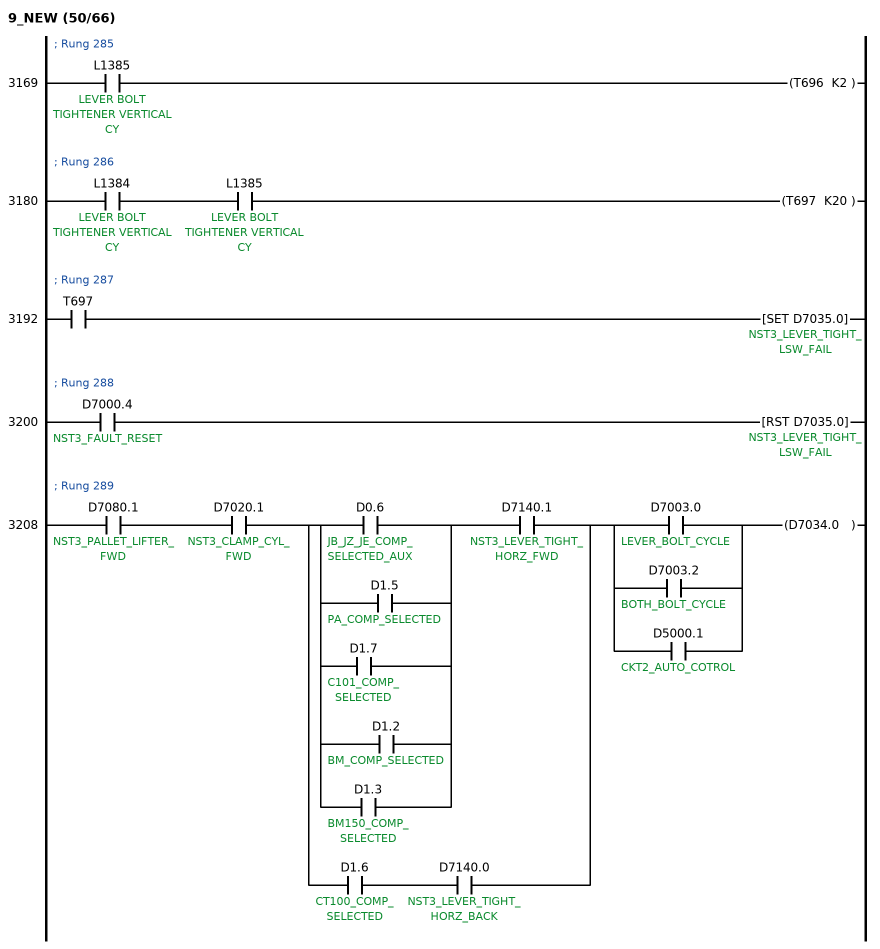
[picture p168: ladder of 9_NEW, rungs at steps 3169 to 3208]
; Rung 285
3169  LD      L1385  ; LEVER BOLT TIGHTENER VERTICAL CY
      OUT     T696 K2
; Rung 286
3180  LD      L1384  ; LEVER BOLT TIGHTENER VERTICAL CY
      AND     L1385  ; LEVER BOLT TIGHTENER VERTICAL CY
      OUT     T697 K20
; Rung 287
3192  LD      T697
      SET     D7035.0  ; NST3_LEVER_TIGHT_LSW_FAIL
; Rung 288
3200  LD      D7000.4  ; NST3_FAULT_RESET
      RST     D7035.0  ; NST3_LEVER_TIGHT_LSW_FAIL
; Rung 289
3208  LD      D7080.1  ; NST3_PALLET_LIFTER_FWD
      AND     D7020.1  ; NST3_CLAMP_CYL_FWD
      LD      D0.6  ; JB_JZ_JE_COMP_SELECTED_AUX
      OR      D1.5  ; PA_COMP_SELECTED
      OR      D1.7  ; C101_COMP_SELECTED
      OR      D1.2  ; BM_COMP_SELECTED
      OR      D1.3  ; BM150_COMP_SELECTED
      AND     D7140.1  ; NST3_LEVER_TIGHT_HORZ_FWD
      LD      D1.6  ; CT100_COMP_SELECTED
      AND     D7140.0  ; NST3_LEVER_TIGHT_HORZ_BACK
      ORB
      ANB
      LD      D7003.0  ; LEVER_BOLT_CYCLE
      OR      D7003.2  ; BOTH_BOLT_CYCLE
      OR      D5000.1  ; CKT2_AUTO_COTROL
      ANB
      OUT     D7034.0
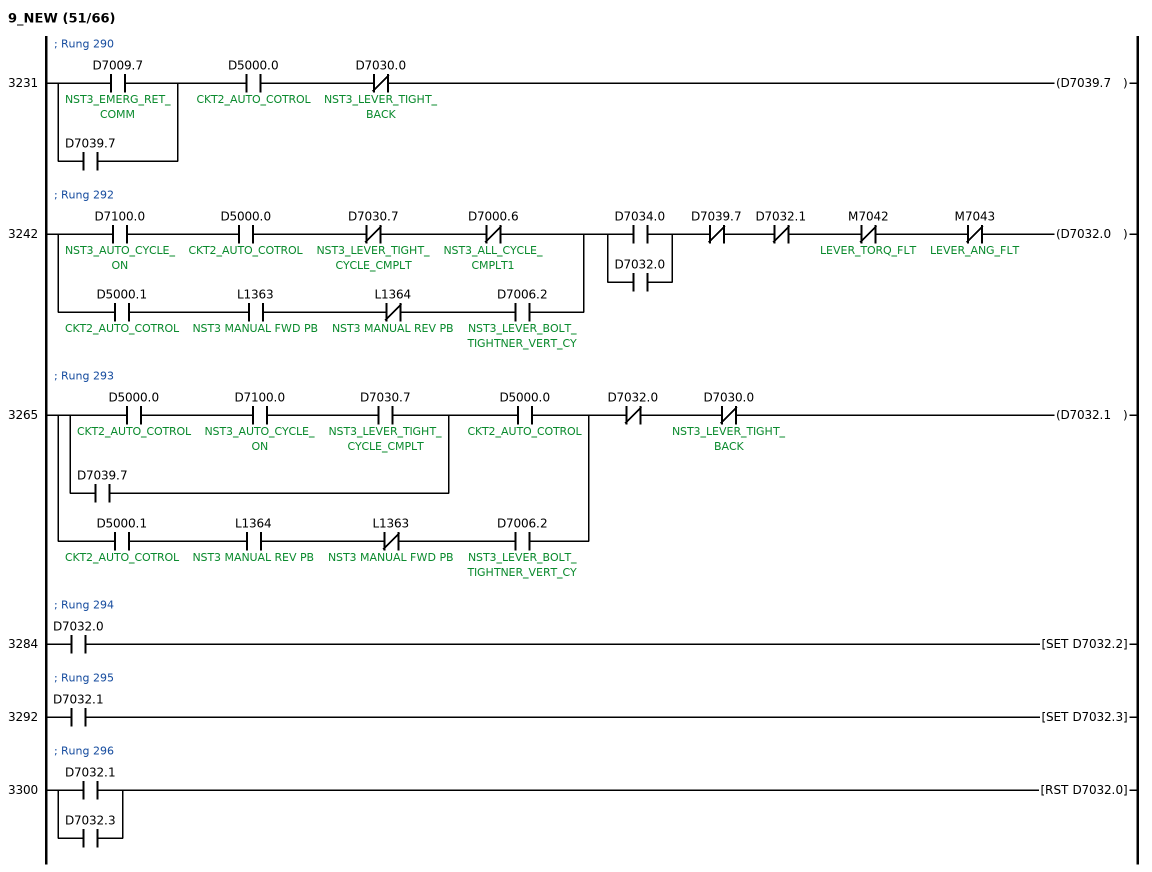
; Rung 290
3231  LD      D7009.7  ; NST3_EMERG_RET_COMM
      OR      D7039.7
      AND     D5000.0  ; CKT2_AUTO_COTROL
      ANI     D7030.0  ; NST3_LEVER_TIGHT_BACK
      OUT     D7039.7
; Rung 292
3242  LD      D7100.0  ; NST3_AUTO_CYCLE_ON
      AND     D5000.0  ; CKT2_AUTO_COTROL
      ANI     D7030.7  ; NST3_LEVER_TIGHT_CYCLE_CMPLT
      ANI     D7000.6  ; NST3_ALL_CYCLE_CMPLT1
      LD      D5000.1  ; CKT2_AUTO_COTROL
      AND     L1363  ; NST3 MANUAL FWD PB
      ANI     L1364  ; NST3 MANUAL REV PB
      AND     D7006.2  ; NST3_LEVER_BOLT_TIGHTNER_VERT_CY
      ORB
      LD      D7034.0
      OR      D7032.0
      ANB
      ANI     D7039.7
      ANI     D7032.1
      ANI     M7042  ; LEVER_TORQ_FLT
      ANI     M7043  ; LEVER_ANG_FLT
      OUT     D7032.0
; Rung 293
3265  LD      D5000.0  ; CKT2_AUTO_COTROL
      AND     D7100.0  ; NST3_AUTO_CYCLE_ON
      AND     D7030.7  ; NST3_LEVER_TIGHT_CYCLE_CMPLT
      OR      D7039.7
      AND     D5000.0  ; CKT2_AUTO_COTROL
      LD      D5000.1  ; CKT2_AUTO_COTROL
      AND     L1364  ; NST3 MANUAL REV PB
      ANI     L1363  ; NST3 MANUAL FWD PB
      AND     D7006.2  ; NST3_LEVER_BOLT_TIGHTNER_VERT_CY
      ORB
      ANI     D7032.0
      ANI     D7030.0  ; NST3_LEVER_TIGHT_BACK
      OUT     D7032.1
; Rung 294
3284  LD      D7032.0
      SET     D7032.2
; Rung 295
3292  LD      D7032.1
      SET     D7032.3
; Rung 296
3300  LD      D7032.1
      OR      D7032.3
      RST     D7032.0
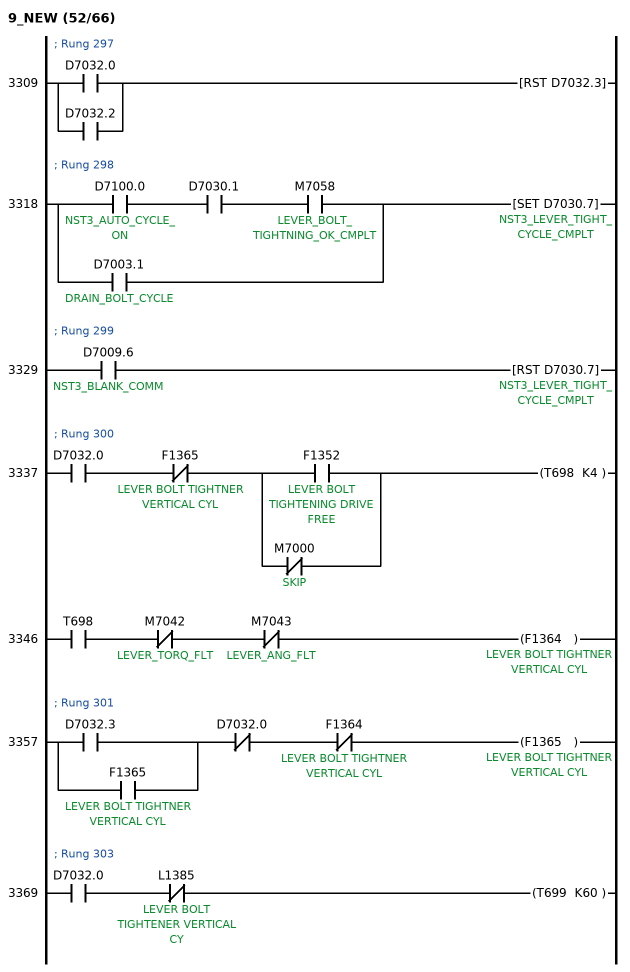
; Rung 297
3309  LD      D7032.0
      OR      D7032.2
      RST     D7032.3
; Rung 298
3318  LD      D7100.0  ; NST3_AUTO_CYCLE_ON
      AND     D7030.1
      AND     M7058  ; LEVER_BOLT_TIGHTNING_OK_CMPLT
      OR      D7003.1  ; DRAIN_BOLT_CYCLE
      SET     D7030.7  ; NST3_LEVER_TIGHT_CYCLE_CMPLT
; Rung 299
3329  LD      D7009.6  ; NST3_BLANK_COMM
      RST     D7030.7  ; NST3_LEVER_TIGHT_CYCLE_CMPLT
; Rung 300
3337  LD      D7032.0
      ANI     F1365  ; LEVER BOLT TIGHTNER VERTICAL CYL
      LD      F1352  ; LEVER BOLT TIGHTENING DRIVE FREE
      ORI     M7000  ; SKIP
      ANB
      OUT     T698 K4
3346  LD      T698
      ANI     M7042  ; LEVER_TORQ_FLT
      ANI     M7043  ; LEVER_ANG_FLT
      OUT     F1364  ; LEVER BOLT TIGHTNER VERTICAL CYL
; Rung 301
3357  LD      D7032.3
      OR      F1365  ; LEVER BOLT TIGHTNER VERTICAL CYL
      ANI     D7032.0
      ANI     F1364  ; LEVER BOLT TIGHTNER VERTICAL CYL
      OUT     F1365  ; LEVER BOLT TIGHTNER VERTICAL CYL
; Rung 303
3369  LD      D7032.0
      ANI     L1385  ; LEVER BOLT TIGHTENER VERTICAL CY
      OUT     T699 K60
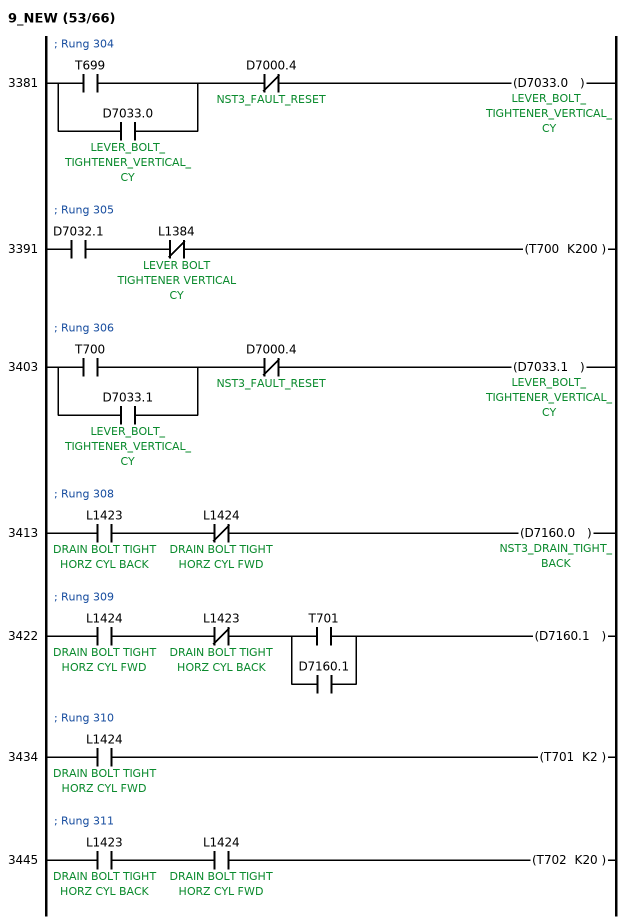
; Rung 304
3381  LD      T699
      OR      D7033.0  ; LEVER_BOLT_TIGHTENER_VERTICAL_CY
      ANI     D7000.4  ; NST3_FAULT_RESET
      OUT     D7033.0  ; LEVER_BOLT_TIGHTENER_VERTICAL_CY
; Rung 305
3391  LD      D7032.1
      ANI     L1384  ; LEVER BOLT TIGHTENER VERTICAL CY
      OUT     T700 K200
; Rung 306
3403  LD      T700
      OR      D7033.1  ; LEVER_BOLT_TIGHTENER_VERTICAL_CY
      ANI     D7000.4  ; NST3_FAULT_RESET
      OUT     D7033.1  ; LEVER_BOLT_TIGHTENER_VERTICAL_CY
; Rung 308
3413  LD      L1423  ; DRAIN BOLT TIGHT HORZ CYL BACK
      ANI     L1424  ; DRAIN BOLT TIGHT HORZ CYL FWD
      OUT     D7160.0  ; NST3_DRAIN_TIGHT_BACK
; Rung 309
3422  LD      L1424  ; DRAIN BOLT TIGHT HORZ CYL FWD
      ANI     L1423  ; DRAIN BOLT TIGHT HORZ CYL BACK
      LD      T701
      OR      D7160.1
      ANB
      OUT     D7160.1
; Rung 310
3434  LD      L1424  ; DRAIN BOLT TIGHT HORZ CYL FWD
      OUT     T701 K2
; Rung 311
3445  LD      L1423  ; DRAIN BOLT TIGHT HORZ CYL BACK
      AND     L1424  ; DRAIN BOLT TIGHT HORZ CYL FWD
      OUT     T702 K20
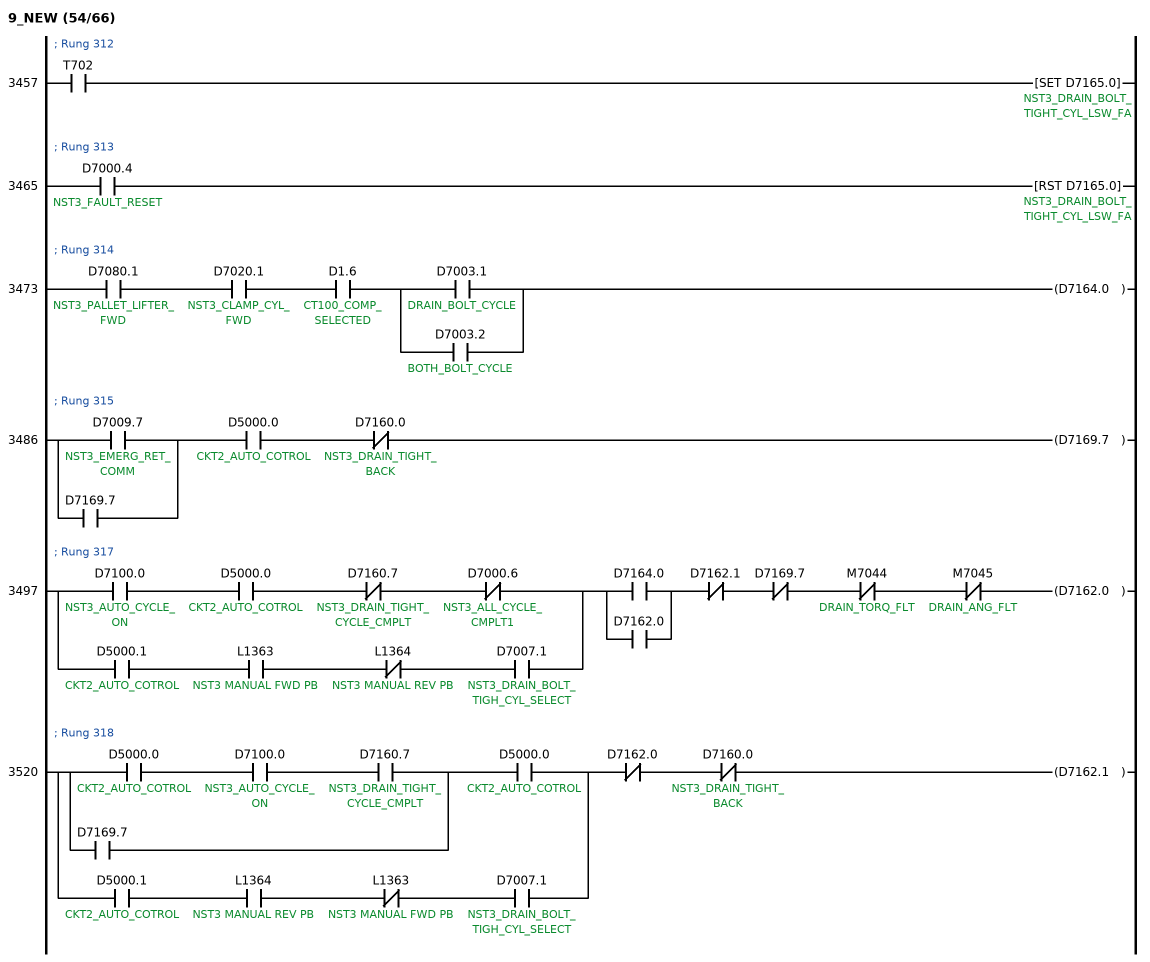
; Rung 312
3457  LD      T702
      SET     D7165.0  ; NST3_DRAIN_BOLT_TIGHT_CYL_LSW_FA
; Rung 313
3465  LD      D7000.4  ; NST3_FAULT_RESET
      RST     D7165.0  ; NST3_DRAIN_BOLT_TIGHT_CYL_LSW_FA
; Rung 314
3473  LD      D7080.1  ; NST3_PALLET_LIFTER_FWD
      AND     D7020.1  ; NST3_CLAMP_CYL_FWD
      AND     D1.6  ; CT100_COMP_SELECTED
      LD      D7003.1  ; DRAIN_BOLT_CYCLE
      OR      D7003.2  ; BOTH_BOLT_CYCLE
      ANB
      OUT     D7164.0
; Rung 315
3486  LD      D7009.7  ; NST3_EMERG_RET_COMM
      OR      D7169.7
      AND     D5000.0  ; CKT2_AUTO_COTROL
      ANI     D7160.0  ; NST3_DRAIN_TIGHT_BACK
      OUT     D7169.7
; Rung 317
3497  LD      D7100.0  ; NST3_AUTO_CYCLE_ON
      AND     D5000.0  ; CKT2_AUTO_COTROL
      ANI     D7160.7  ; NST3_DRAIN_TIGHT_CYCLE_CMPLT
      ANI     D7000.6  ; NST3_ALL_CYCLE_CMPLT1
      LD      D5000.1  ; CKT2_AUTO_COTROL
      AND     L1363  ; NST3 MANUAL FWD PB
      ANI     L1364  ; NST3 MANUAL REV PB
      AND     D7007.1  ; NST3_DRAIN_BOLT_TIGH_CYL_SELECT
      ORB
      LD      D7164.0
      OR      D7162.0
      ANB
      ANI     D7162.1
      ANI     D7169.7
      ANI     M7044  ; DRAIN_TORQ_FLT
      ANI     M7045  ; DRAIN_ANG_FLT
      OUT     D7162.0
; Rung 318
3520  LD      D5000.0  ; CKT2_AUTO_COTROL
      AND     D7100.0  ; NST3_AUTO_CYCLE_ON
      AND     D7160.7  ; NST3_DRAIN_TIGHT_CYCLE_CMPLT
      OR      D7169.7
      AND     D5000.0  ; CKT2_AUTO_COTROL
      LD      D5000.1  ; CKT2_AUTO_COTROL
      AND     L1364  ; NST3 MANUAL REV PB
      ANI     L1363  ; NST3 MANUAL FWD PB
      AND     D7007.1  ; NST3_DRAIN_BOLT_TIGH_CYL_SELECT
      ORB
      ANI     D7162.0
      ANI     D7160.0  ; NST3_DRAIN_TIGHT_BACK
      OUT     D7162.1
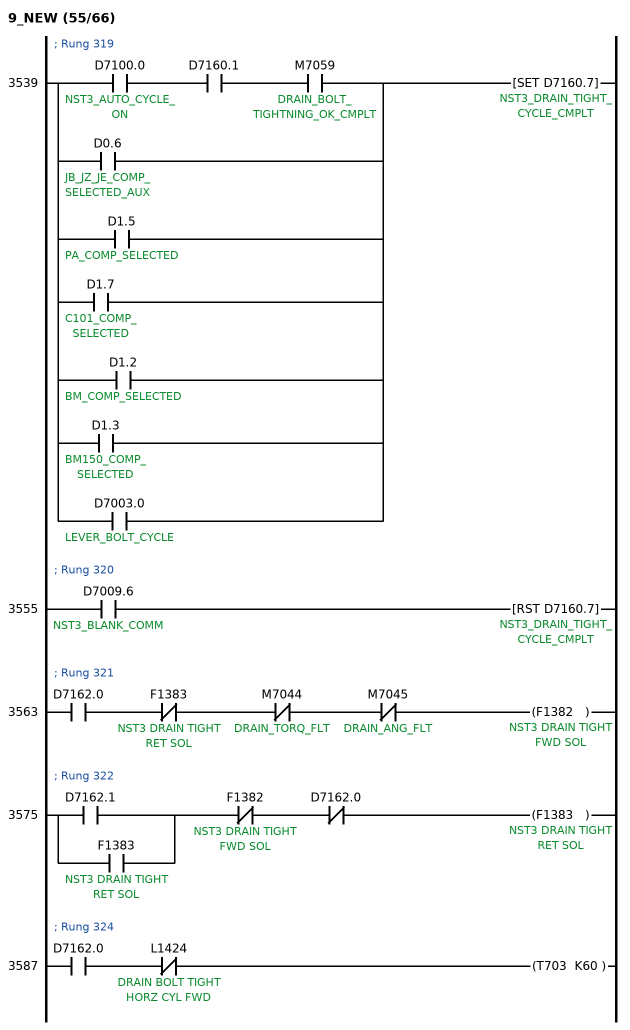
; Rung 319
3539  LD      D7100.0  ; NST3_AUTO_CYCLE_ON
      AND     D7160.1
      AND     M7059  ; DRAIN_BOLT_TIGHTNING_OK_CMPLT
      OR      D0.6  ; JB_JZ_JE_COMP_SELECTED_AUX
      OR      D1.5  ; PA_COMP_SELECTED
      OR      D1.7  ; C101_COMP_SELECTED
      OR      D1.2  ; BM_COMP_SELECTED
      OR      D1.3  ; BM150_COMP_SELECTED
      OR      D7003.0  ; LEVER_BOLT_CYCLE
      SET     D7160.7  ; NST3_DRAIN_TIGHT_CYCLE_CMPLT
; Rung 320
3555  LD      D7009.6  ; NST3_BLANK_COMM
      RST     D7160.7  ; NST3_DRAIN_TIGHT_CYCLE_CMPLT
; Rung 321
3563  LD      D7162.0
      ANI     F1383  ; NST3 DRAIN TIGHT RET SOL
      ANI     M7044  ; DRAIN_TORQ_FLT
      ANI     M7045  ; DRAIN_ANG_FLT
      OUT     F1382  ; NST3 DRAIN TIGHT FWD SOL
; Rung 322
3575  LD      D7162.1
      OR      F1383  ; NST3 DRAIN TIGHT RET SOL
      ANI     F1382  ; NST3 DRAIN TIGHT FWD SOL
      ANI     D7162.0
      OUT     F1383  ; NST3 DRAIN TIGHT RET SOL
; Rung 324
3587  LD      D7162.0
      ANI     L1424  ; DRAIN BOLT TIGHT HORZ CYL FWD
      OUT     T703 K60
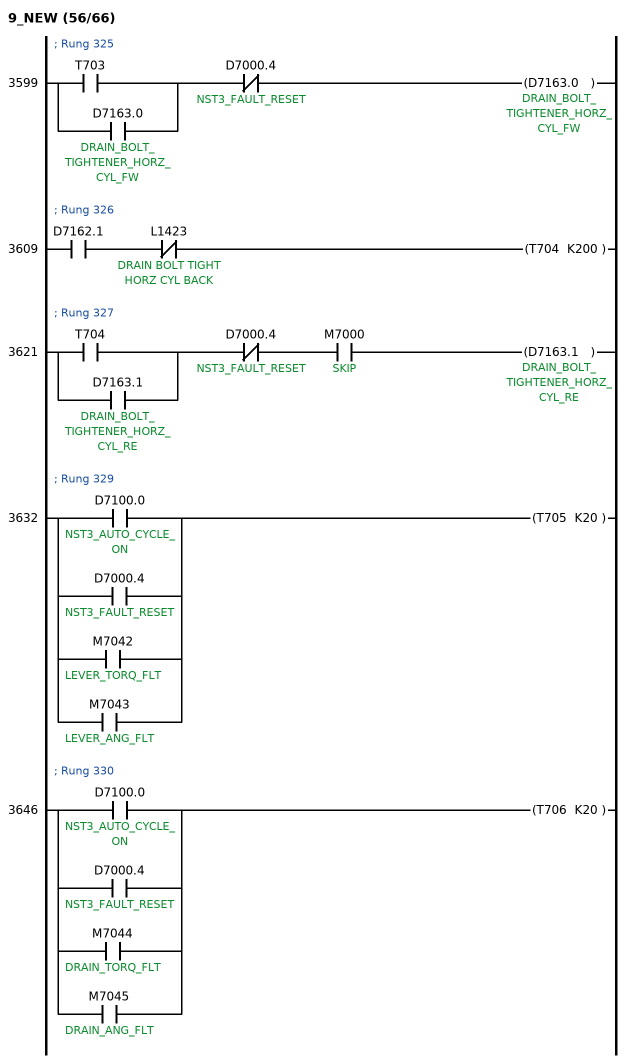
; Rung 325
3599  LD      T703
      OR      D7163.0  ; DRAIN_BOLT_TIGHTENER_HORZ_CYL_FW
      ANI     D7000.4  ; NST3_FAULT_RESET
      OUT     D7163.0  ; DRAIN_BOLT_TIGHTENER_HORZ_CYL_FW
; Rung 326
3609  LD      D7162.1
      ANI     L1423  ; DRAIN BOLT TIGHT HORZ CYL BACK
      OUT     T704 K200
; Rung 327
3621  LD      T704
      OR      D7163.1  ; DRAIN_BOLT_TIGHTENER_HORZ_CYL_RE
      ANI     D7000.4  ; NST3_FAULT_RESET
      AND     M7000  ; SKIP
      OUT     D7163.1  ; DRAIN_BOLT_TIGHTENER_HORZ_CYL_RE
; Rung 329
3632  LD      D7100.0  ; NST3_AUTO_CYCLE_ON
      OR      D7000.4  ; NST3_FAULT_RESET
      OR      M7042  ; LEVER_TORQ_FLT
      OR      M7043  ; LEVER_ANG_FLT
      OUT     T705 K20
; Rung 330
3646  LD      D7100.0  ; NST3_AUTO_CYCLE_ON
      OR      D7000.4  ; NST3_FAULT_RESET
      OR      M7044  ; DRAIN_TORQ_FLT
      OR      M7045  ; DRAIN_ANG_FLT
      OUT     T706 K20
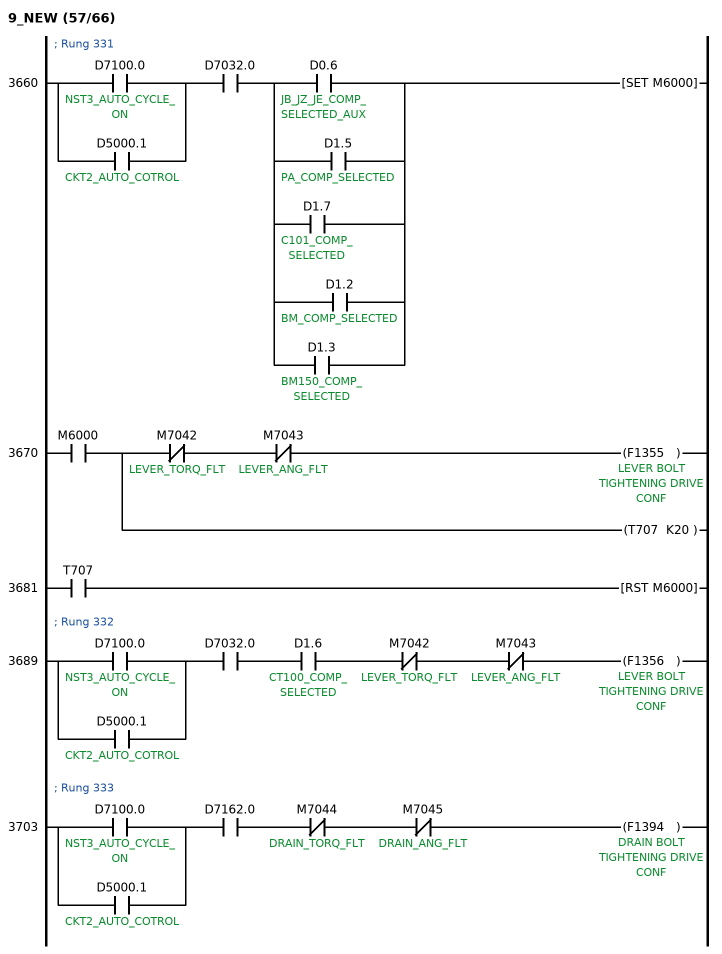
; Rung 331
3660  LD      D7100.0  ; NST3_AUTO_CYCLE_ON
      OR      D5000.1  ; CKT2_AUTO_COTROL
      AND     D7032.0
      LD      D0.6  ; JB_JZ_JE_COMP_SELECTED_AUX
      OR      D1.5  ; PA_COMP_SELECTED
      OR      D1.7  ; C101_COMP_SELECTED
      OR      D1.2  ; BM_COMP_SELECTED
      OR      D1.3  ; BM150_COMP_SELECTED
      ANB
      SET     M6000
3670  LD      M6000
      MPS
      ANI     M7042  ; LEVER_TORQ_FLT
      ANI     M7043  ; LEVER_ANG_FLT
      OUT     F1355  ; LEVER BOLT TIGHTENING DRIVE CONF
      MPP
      OUT     T707 K20
3681  LD      T707
      RST     M6000
; Rung 332
3689  LD      D7100.0  ; NST3_AUTO_CYCLE_ON
      OR      D5000.1  ; CKT2_AUTO_COTROL
      AND     D7032.0
      AND     D1.6  ; CT100_COMP_SELECTED
      ANI     M7042  ; LEVER_TORQ_FLT
      ANI     M7043  ; LEVER_ANG_FLT
      OUT     F1356  ; LEVER BOLT TIGHTENING DRIVE CONF
; Rung 333
3703  LD      D7100.0  ; NST3_AUTO_CYCLE_ON
      OR      D5000.1  ; CKT2_AUTO_COTROL
      AND     D7162.0
      ANI     M7044  ; DRAIN_TORQ_FLT
      ANI     M7045  ; DRAIN_ANG_FLT
      OUT     F1394  ; DRAIN BOLT TIGHTENING DRIVE CONF
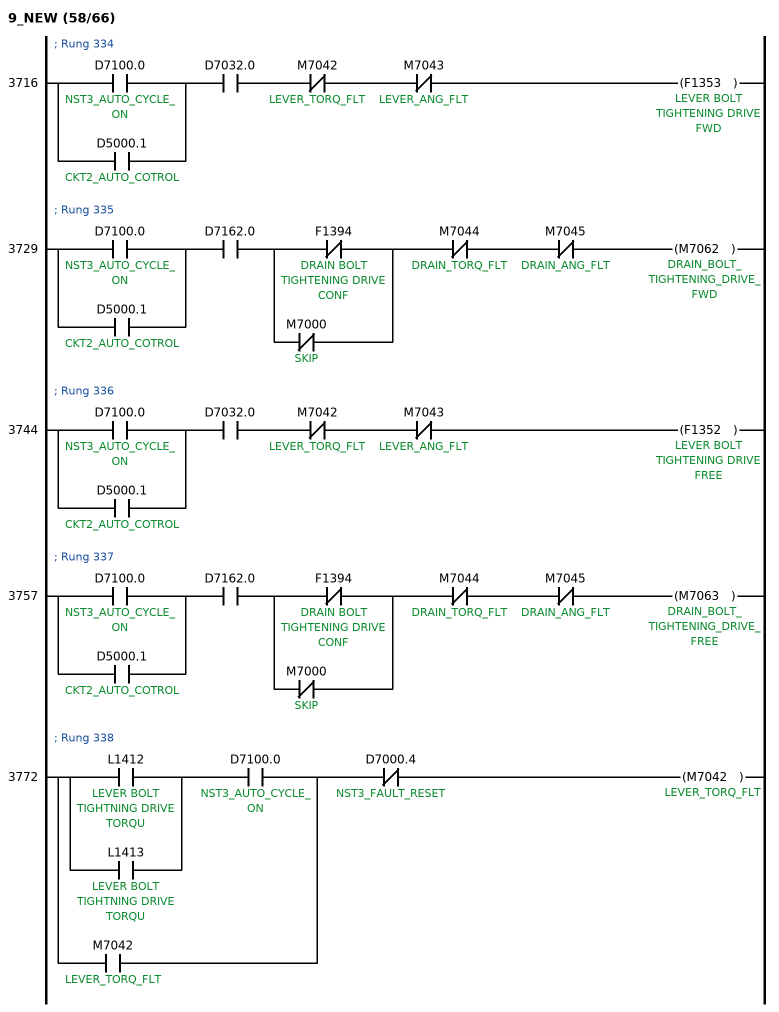
; Rung 334
3716  LD      D7100.0  ; NST3_AUTO_CYCLE_ON
      OR      D5000.1  ; CKT2_AUTO_COTROL
      AND     D7032.0
      ANI     M7042  ; LEVER_TORQ_FLT
      ANI     M7043  ; LEVER_ANG_FLT
      OUT     F1353  ; LEVER BOLT TIGHTENING DRIVE FWD
; Rung 335
3729  LD      D7100.0  ; NST3_AUTO_CYCLE_ON
      OR      D5000.1  ; CKT2_AUTO_COTROL
      AND     D7162.0
      LDI     F1394  ; DRAIN BOLT TIGHTENING DRIVE CONF
      ORI     M7000  ; SKIP
      ANB
      ANI     M7044  ; DRAIN_TORQ_FLT
      ANI     M7045  ; DRAIN_ANG_FLT
      OUT     M7062  ; DRAIN_BOLT_TIGHTENING_DRIVE_FWD
; Rung 336
3744  LD      D7100.0  ; NST3_AUTO_CYCLE_ON
      OR      D5000.1  ; CKT2_AUTO_COTROL
      AND     D7032.0
      ANI     M7042  ; LEVER_TORQ_FLT
      ANI     M7043  ; LEVER_ANG_FLT
      OUT     F1352  ; LEVER BOLT TIGHTENING DRIVE FREE
; Rung 337
3757  LD      D7100.0  ; NST3_AUTO_CYCLE_ON
      OR      D5000.1  ; CKT2_AUTO_COTROL
      AND     D7162.0
      LDI     F1394  ; DRAIN BOLT TIGHTENING DRIVE CONF
      ORI     M7000  ; SKIP
      ANB
      ANI     M7044  ; DRAIN_TORQ_FLT
      ANI     M7045  ; DRAIN_ANG_FLT
      OUT     M7063  ; DRAIN_BOLT_TIGHTENING_DRIVE_FREE
; Rung 338
3772  LD      L1412  ; LEVER BOLT TIGHTNING DRIVE TORQU
      OR      L1413  ; LEVER BOLT TIGHTNING DRIVE TORQU
      AND     D7100.0  ; NST3_AUTO_CYCLE_ON
      OR      M7042  ; LEVER_TORQ_FLT
      ANI     D7000.4  ; NST3_FAULT_RESET
      OUT     M7042  ; LEVER_TORQ_FLT
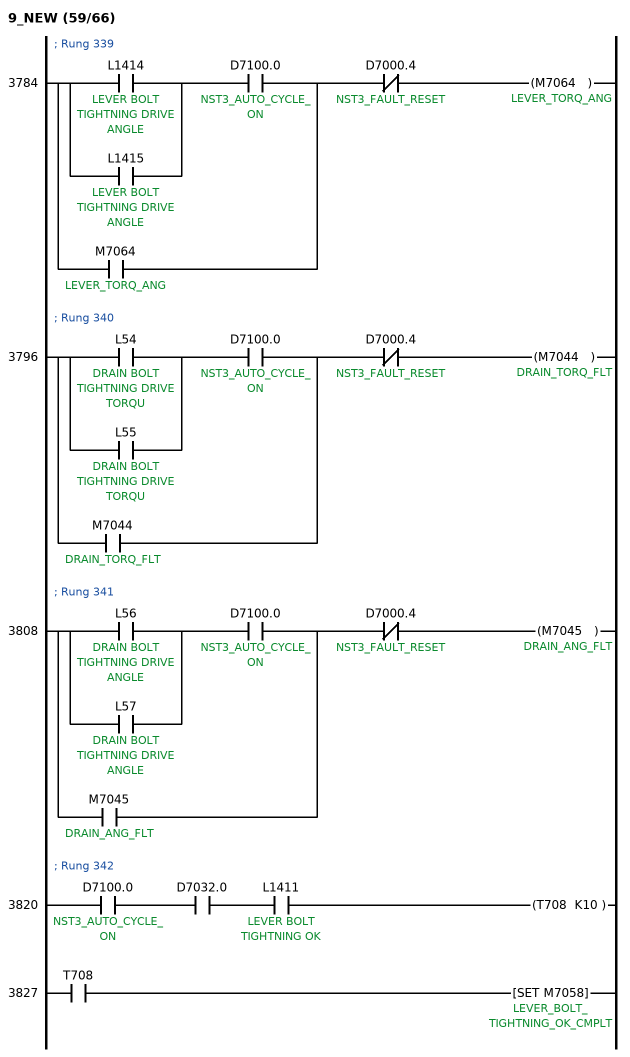
; Rung 339
3784  LD      L1414  ; LEVER BOLT TIGHTNING DRIVE ANGLE
      OR      L1415  ; LEVER BOLT TIGHTNING DRIVE ANGLE
      AND     D7100.0  ; NST3_AUTO_CYCLE_ON
      OR      M7064  ; LEVER_TORQ_ANG
      ANI     D7000.4  ; NST3_FAULT_RESET
      OUT     M7064  ; LEVER_TORQ_ANG
; Rung 340
3796  LD      L54  ; DRAIN BOLT TIGHTNING DRIVE TORQU
      OR      L55  ; DRAIN BOLT TIGHTNING DRIVE TORQU
      AND     D7100.0  ; NST3_AUTO_CYCLE_ON
      OR      M7044  ; DRAIN_TORQ_FLT
      ANI     D7000.4  ; NST3_FAULT_RESET
      OUT     M7044  ; DRAIN_TORQ_FLT
; Rung 341
3808  LD      L56  ; DRAIN BOLT TIGHTNING DRIVE ANGLE
      OR      L57  ; DRAIN BOLT TIGHTNING DRIVE ANGLE
      AND     D7100.0  ; NST3_AUTO_CYCLE_ON
      OR      M7045  ; DRAIN_ANG_FLT
      ANI     D7000.4  ; NST3_FAULT_RESET
      OUT     M7045  ; DRAIN_ANG_FLT
; Rung 342
3820  LD      D7100.0  ; NST3_AUTO_CYCLE_ON
      AND     D7032.0
      AND     L1411  ; LEVER BOLT TIGHTNING OK
      OUT     T708 K10
3827  LD      T708
      SET     M7058  ; LEVER_BOLT_TIGHTNING_OK_CMPLT
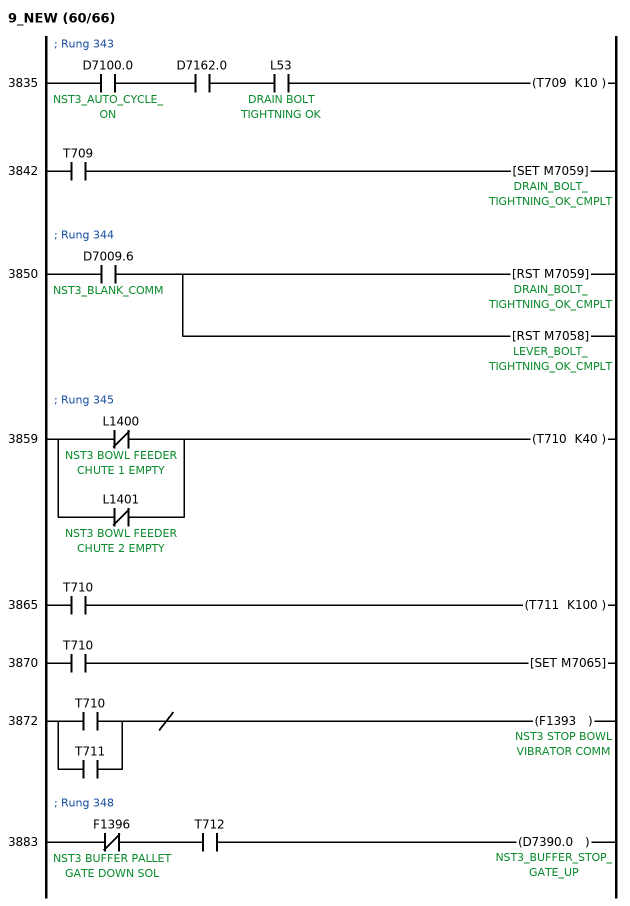
; Rung 343
3835  LD      D7100.0  ; NST3_AUTO_CYCLE_ON
      AND     D7162.0
      AND     L53  ; DRAIN BOLT TIGHTNING OK
      OUT     T709 K10
3842  LD      T709
      SET     M7059  ; DRAIN_BOLT_TIGHTNING_OK_CMPLT
; Rung 344
3850  LD      D7009.6  ; NST3_BLANK_COMM
      RST     M7059  ; DRAIN_BOLT_TIGHTNING_OK_CMPLT
      RST     M7058  ; LEVER_BOLT_TIGHTNING_OK_CMPLT
; Rung 345
3859  LDI     L1400  ; NST3 BOWL FEEDER CHUTE 1 EMPTY
      ORI     L1401  ; NST3 BOWL FEEDER CHUTE 2 EMPTY
      OUT     T710 K40
3865  LD      T710
      OUT     T711 K100
3870  LD      T710
      SET     M7065
3872  LD      T710
      OR      T711
      INV
      OUT     F1393  ; NST3 STOP BOWL VIBRATOR COMM
; Rung 348
3883  LDI     F1396  ; NST3 BUFFER PALLET GATE DOWN SOL
      AND     T712
      OUT     D7390.0  ; NST3_BUFFER_STOP_GATE_UP
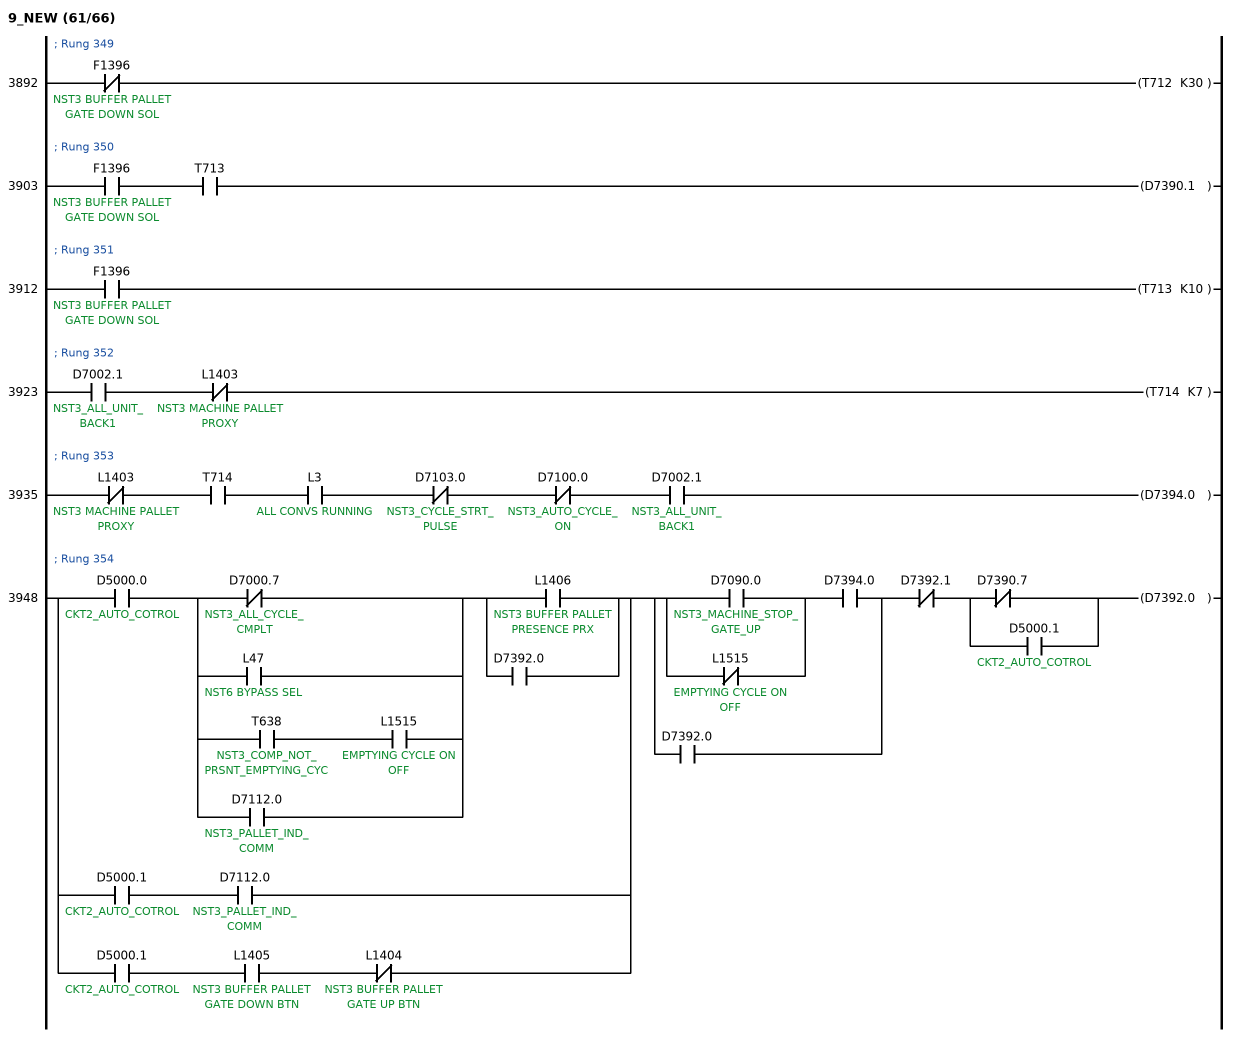
; Rung 349
3892  LDI     F1396  ; NST3 BUFFER PALLET GATE DOWN SOL
      OUT     T712 K30
; Rung 350
3903  LD      F1396  ; NST3 BUFFER PALLET GATE DOWN SOL
      AND     T713
      OUT     D7390.1
; Rung 351
3912  LD      F1396  ; NST3 BUFFER PALLET GATE DOWN SOL
      OUT     T713 K10
; Rung 352
3923  LD      D7002.1  ; NST3_ALL_UNIT_BACK1
      ANI     L1403  ; NST3 MACHINE PALLET PROXY
      OUT     T714 K7
; Rung 353
3935  LDI     L1403  ; NST3 MACHINE PALLET PROXY
      AND     T714
      AND     L3  ; ALL CONVS RUNNING
      ANI     D7103.0  ; NST3_CYCLE_STRT_PULSE
      ANI     D7100.0  ; NST3_AUTO_CYCLE_ON
      AND     D7002.1  ; NST3_ALL_UNIT_BACK1
      OUT     D7394.0
; Rung 354
3948  LD      D5000.0  ; CKT2_AUTO_COTROL
      LDI     D7000.7  ; NST3_ALL_CYCLE_CMPLT
      OR      L47  ; NST6 BYPASS SEL
      LD      T638  ; NST3_COMP_NOT_PRSNT_EMPTYING_CYC
      AND     L1515  ; EMPTYING CYCLE ON OFF
      ORB
      OR      D7112.0  ; NST3_PALLET_IND_COMM
      ANB
      LD      L1406  ; NST3 BUFFER PALLET PRESENCE PRX
      OR      D7392.0
      ANB
      LD      D5000.1  ; CKT2_AUTO_COTROL
      AND     D7112.0  ; NST3_PALLET_IND_COMM
      ORB
      LD      D5000.1  ; CKT2_AUTO_COTROL
      AND     L1405  ; NST3 BUFFER PALLET GATE DOWN BTN
      ANI     L1404  ; NST3 BUFFER PALLET GATE UP BTN
      ORB
      LD      D7090.0  ; NST3_MACHINE_STOP_GATE_UP
      ORI     L1515  ; EMPTYING CYCLE ON OFF
      AND     D7394.0
      OR      D7392.0
      ANB
      ANI     D7392.1
      LDI     D7390.7
      OR      D5000.1  ; CKT2_AUTO_COTROL
      ANB
      OUT     D7392.0
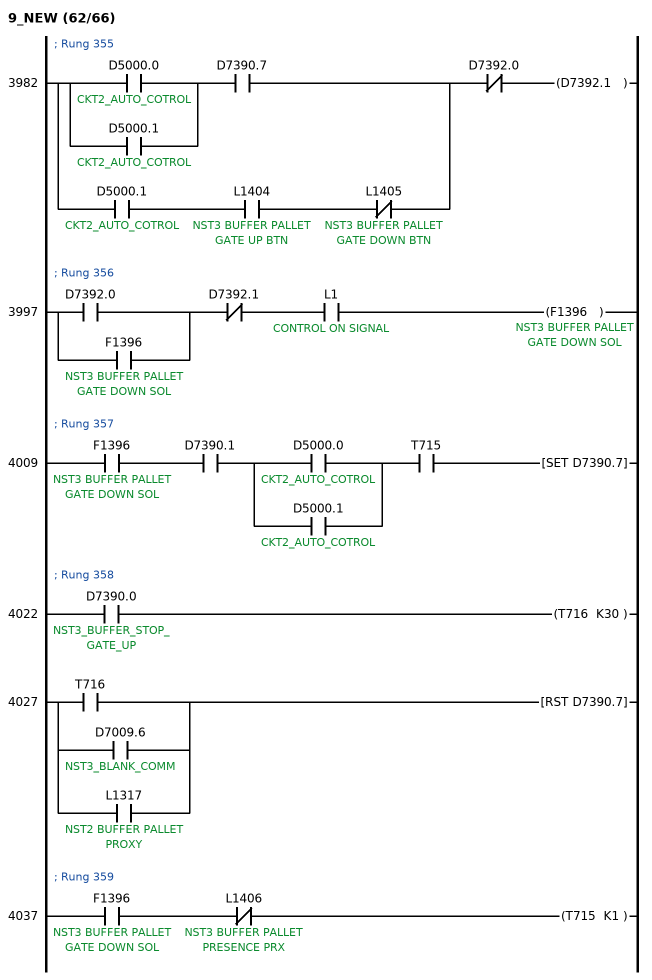
; Rung 355
3982  LD      D5000.0  ; CKT2_AUTO_COTROL
      OR      D5000.1  ; CKT2_AUTO_COTROL
      AND     D7390.7
      LD      D5000.1  ; CKT2_AUTO_COTROL
      AND     L1404  ; NST3 BUFFER PALLET GATE UP BTN
      ANI     L1405  ; NST3 BUFFER PALLET GATE DOWN BTN
      ORB
      ANI     D7392.0
      OUT     D7392.1
; Rung 356
3997  LD      D7392.0
      OR      F1396  ; NST3 BUFFER PALLET GATE DOWN SOL
      ANI     D7392.1
      AND     L1  ; CONTROL ON SIGNAL
      OUT     F1396  ; NST3 BUFFER PALLET GATE DOWN SOL
; Rung 357
4009  LD      F1396  ; NST3 BUFFER PALLET GATE DOWN SOL
      AND     D7390.1
      LD      D5000.0  ; CKT2_AUTO_COTROL
      OR      D5000.1  ; CKT2_AUTO_COTROL
      ANB
      AND     T715
      SET     D7390.7
; Rung 358
4022  LD      D7390.0  ; NST3_BUFFER_STOP_GATE_UP
      OUT     T716 K30
4027  LD      T716
      OR      D7009.6  ; NST3_BLANK_COMM
      OR      L1317  ; NST2 BUFFER PALLET PROXY
      RST     D7390.7
; Rung 359
4037  LD      F1396  ; NST3 BUFFER PALLET GATE DOWN SOL
      ANI     L1406  ; NST3 BUFFER PALLET PRESENCE PRX
      OUT     T715 K1
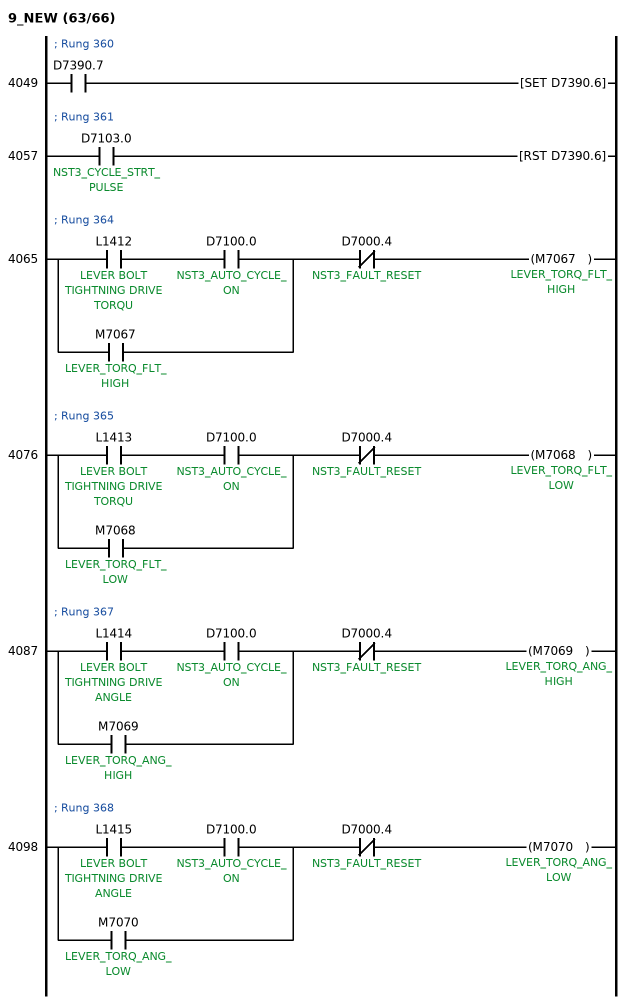
; Rung 360
4049  LD      D7390.7
      SET     D7390.6
; Rung 361
4057  LD      D7103.0  ; NST3_CYCLE_STRT_PULSE
      RST     D7390.6
; Rung 364
4065  LD      L1412  ; LEVER BOLT TIGHTNING DRIVE TORQU
      AND     D7100.0  ; NST3_AUTO_CYCLE_ON
      OR      M7067  ; LEVER_TORQ_FLT_HIGH
      ANI     D7000.4  ; NST3_FAULT_RESET
      OUT     M7067  ; LEVER_TORQ_FLT_HIGH
; Rung 365
4076  LD      L1413  ; LEVER BOLT TIGHTNING DRIVE TORQU
      AND     D7100.0  ; NST3_AUTO_CYCLE_ON
      OR      M7068  ; LEVER_TORQ_FLT_LOW
      ANI     D7000.4  ; NST3_FAULT_RESET
      OUT     M7068  ; LEVER_TORQ_FLT_LOW
; Rung 367
4087  LD      L1414  ; LEVER BOLT TIGHTNING DRIVE ANGLE
      AND     D7100.0  ; NST3_AUTO_CYCLE_ON
      OR      M7069  ; LEVER_TORQ_ANG_HIGH
      ANI     D7000.4  ; NST3_FAULT_RESET
      OUT     M7069  ; LEVER_TORQ_ANG_HIGH
; Rung 368
4098  LD      L1415  ; LEVER BOLT TIGHTNING DRIVE ANGLE
      AND     D7100.0  ; NST3_AUTO_CYCLE_ON
      OR      M7070  ; LEVER_TORQ_ANG_LOW
      ANI     D7000.4  ; NST3_FAULT_RESET
      OUT     M7070  ; LEVER_TORQ_ANG_LOW
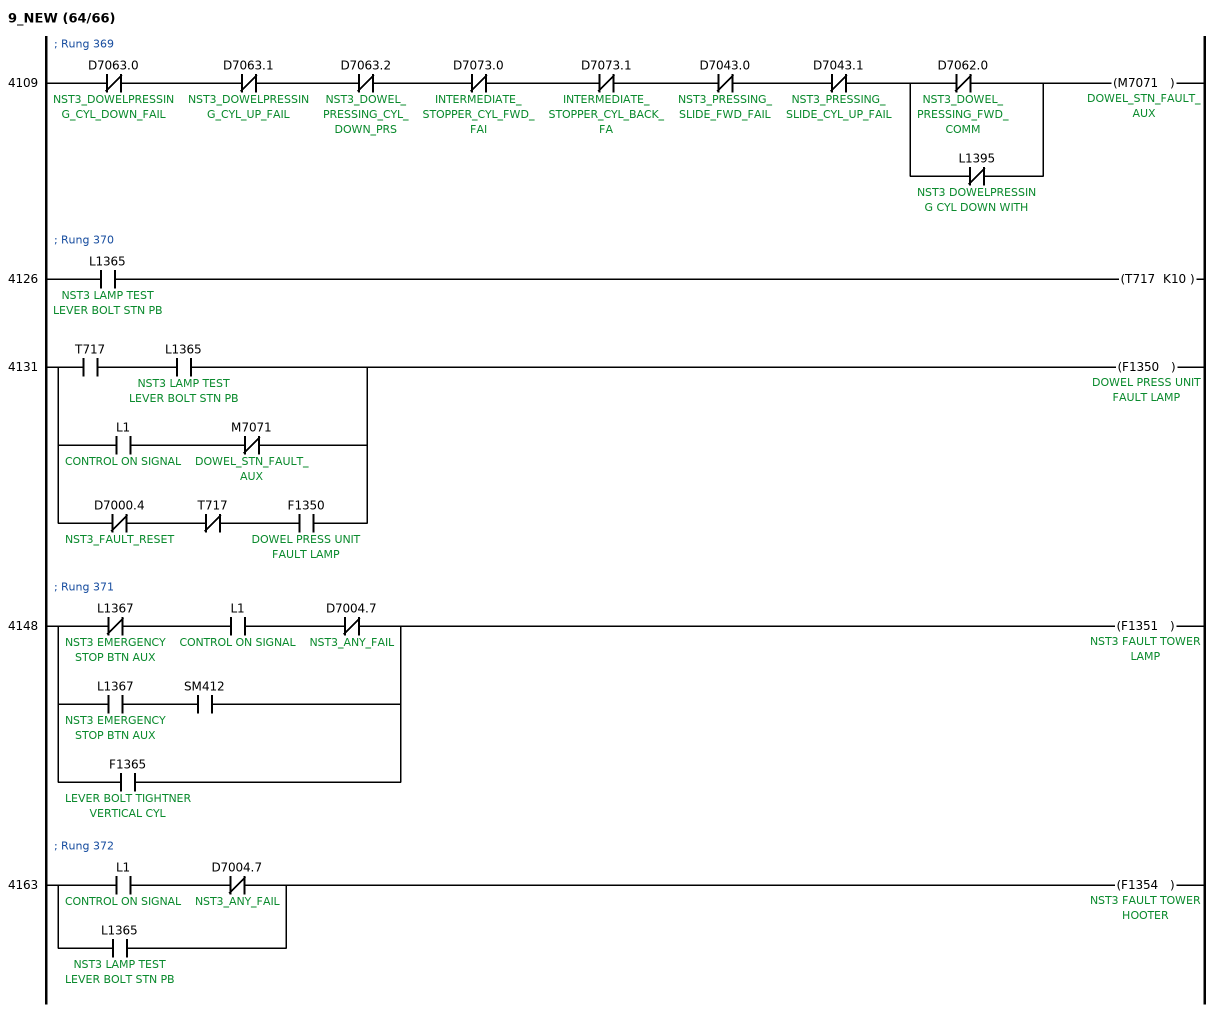
; Rung 369
4109  LDI     D7063.0  ; NST3_DOWELPRESSING_CYL_DOWN_FAIL
      ANI     D7063.1  ; NST3_DOWELPRESSING_CYL_UP_FAIL
      ANI     D7063.2  ; NST3_DOWEL_PRESSING_CYL_DOWN_PRS
      ANI     D7073.0  ; INTERMEDIATE_STOPPER_CYL_FWD_FAI
      ANI     D7073.1  ; INTERMEDIATE_STOPPER_CYL_BACK_FA
      ANI     D7043.0  ; NST3_PRESSING_SLIDE_FWD_FAIL
      ANI     D7043.1  ; NST3_PRESSING_SLIDE_CYL_UP_FAIL
      LDI     D7062.0  ; NST3_DOWEL_PRESSING_FWD_COMM
      ORI     L1395  ; NST3 DOWELPRESSING CYL DOWN WITH
      ANB
      OUT     M7071  ; DOWEL_STN_FAULT_AUX
; Rung 370
4126  LD      L1365  ; NST3 LAMP TEST LEVER BOLT STN PB
      OUT     T717 K10
4131  LD      T717
      AND     L1365  ; NST3 LAMP TEST LEVER BOLT STN PB
      LD      L1  ; CONTROL ON SIGNAL
      ANI     M7071  ; DOWEL_STN_FAULT_AUX
      ORB
      LDI     D7000.4  ; NST3_FAULT_RESET
      ANI     T717
      AND     F1350  ; DOWEL PRESS UNIT FAULT LAMP
      ORB
      OUT     F1350  ; DOWEL PRESS UNIT FAULT LAMP
; Rung 371
4148  LDI     L1367  ; NST3 EMERGENCY STOP BTN AUX
      AND     L1  ; CONTROL ON SIGNAL
      ANI     D7004.7  ; NST3_ANY_FAIL
      LD      L1367  ; NST3 EMERGENCY STOP BTN AUX
      AND     SM412
      ORB
      OR      F1365  ; LEVER BOLT TIGHTNER VERTICAL CYL
      OUT     F1351  ; NST3 FAULT TOWER LAMP
; Rung 372
4163  LD      L1  ; CONTROL ON SIGNAL
      ANI     D7004.7  ; NST3_ANY_FAIL
      OR      L1365  ; NST3 LAMP TEST LEVER BOLT STN PB
      OUT     F1354  ; NST3 FAULT TOWER HOOTER
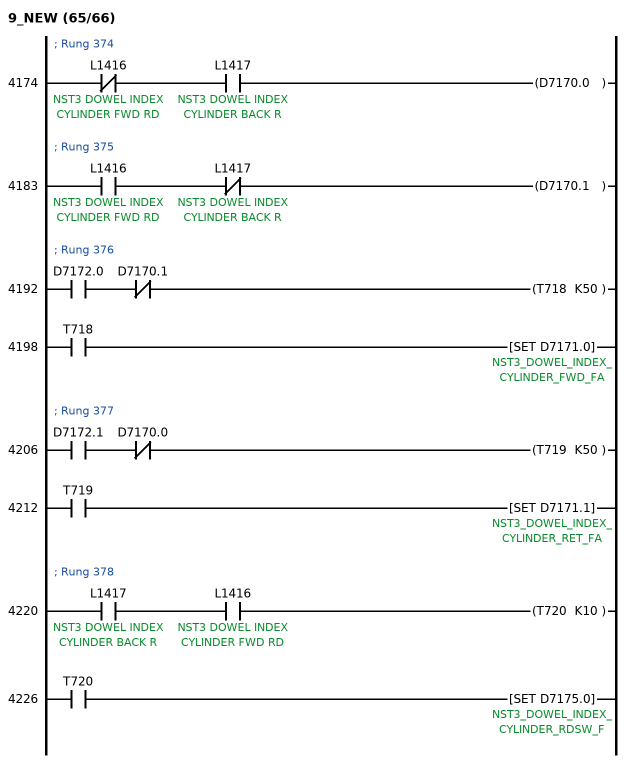
; Rung 374
4174  LDI     L1416  ; NST3 DOWEL INDEX CYLINDER FWD RD
      AND     L1417  ; NST3 DOWEL INDEX CYLINDER BACK R
      OUT     D7170.0
; Rung 375
4183  LD      L1416  ; NST3 DOWEL INDEX CYLINDER FWD RD
      ANI     L1417  ; NST3 DOWEL INDEX CYLINDER BACK R
      OUT     D7170.1
; Rung 376
4192  LD      D7172.0
      ANI     D7170.1
      OUT     T718 K50
4198  LD      T718
      SET     D7171.0  ; NST3_DOWEL_INDEX_CYLINDER_FWD_FA
; Rung 377
4206  LD      D7172.1
      ANI     D7170.0
      OUT     T719 K50
4212  LD      T719
      SET     D7171.1  ; NST3_DOWEL_INDEX_CYLINDER_RET_FA
; Rung 378
4220  LD      L1417  ; NST3 DOWEL INDEX CYLINDER BACK R
      AND     L1416  ; NST3 DOWEL INDEX CYLINDER FWD RD
      OUT     T720 K10
4226  LD      T720
      SET     D7175.0  ; NST3_DOWEL_INDEX_CYLINDER_RDSW_F
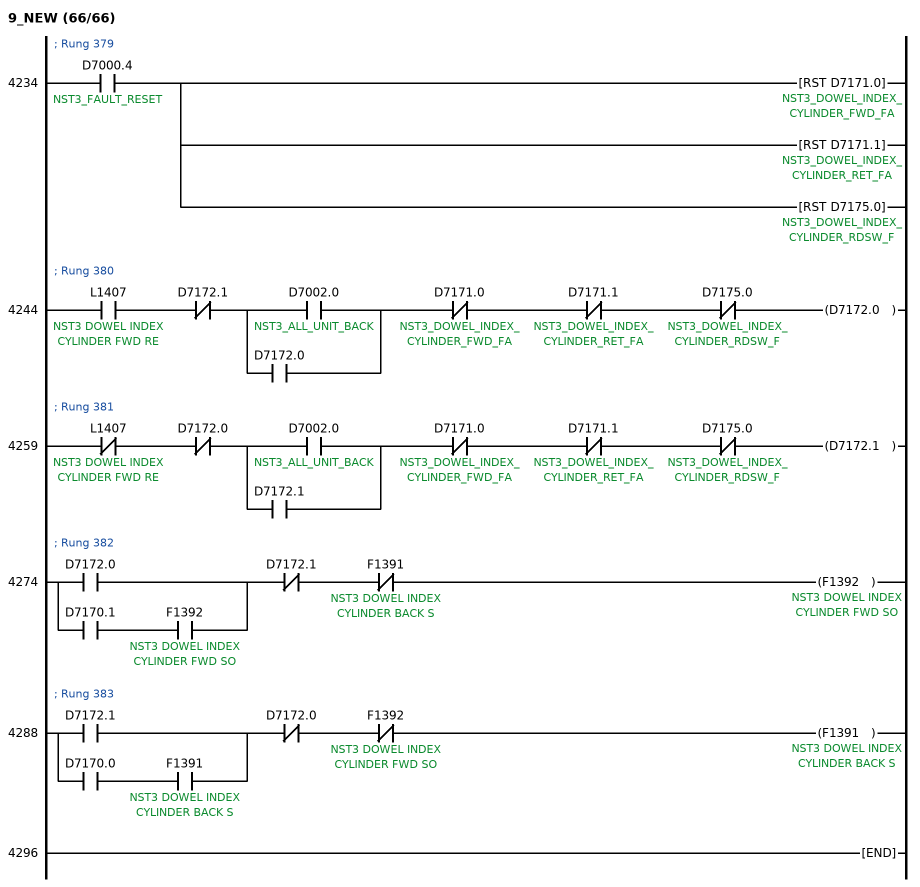
; Rung 379
4234  LD      D7000.4  ; NST3_FAULT_RESET
      RST     D7171.0  ; NST3_DOWEL_INDEX_CYLINDER_FWD_FA
      RST     D7171.1  ; NST3_DOWEL_INDEX_CYLINDER_RET_FA
      RST     D7175.0  ; NST3_DOWEL_INDEX_CYLINDER_RDSW_F
; Rung 380
4244  LD      L1407  ; NST3 DOWEL INDEX CYLINDER FWD RE
      ANI     D7172.1
      LD      D7002.0  ; NST3_ALL_UNIT_BACK
      OR      D7172.0
      ANB
      ANI     D7171.0  ; NST3_DOWEL_INDEX_CYLINDER_FWD_FA
      ANI     D7171.1  ; NST3_DOWEL_INDEX_CYLINDER_RET_FA
      ANI     D7175.0  ; NST3_DOWEL_INDEX_CYLINDER_RDSW_F
      OUT     D7172.0
; Rung 381
4259  LDI     L1407  ; NST3 DOWEL INDEX CYLINDER FWD RE
      ANI     D7172.0
      LD      D7002.0  ; NST3_ALL_UNIT_BACK
      OR      D7172.1
      ANB
      ANI     D7171.0  ; NST3_DOWEL_INDEX_CYLINDER_FWD_FA
      ANI     D7171.1  ; NST3_DOWEL_INDEX_CYLINDER_RET_FA
      ANI     D7175.0  ; NST3_DOWEL_INDEX_CYLINDER_RDSW_F
      OUT     D7172.1
; Rung 382
4274  LD      D7172.0
      LD      D7170.1
      AND     F1392  ; NST3 DOWEL INDEX CYLINDER FWD SO
      ORB
      ANI     D7172.1
      ANI     F1391  ; NST3 DOWEL INDEX CYLINDER BACK S
      OUT     F1392  ; NST3 DOWEL INDEX CYLINDER FWD SO
; Rung 383
4288  LD      D7172.1
      LD      D7170.0
      AND     F1391  ; NST3 DOWEL INDEX CYLINDER BACK S
      ORB
      ANI     D7172.0
      ANI     F1392  ; NST3 DOWEL INDEX CYLINDER FWD SO
      OUT     F1391  ; NST3 DOWEL INDEX CYLINDER BACK S
4296  END
END_PROGRAM

PROGRAM 10_NEW  // ST4 CK2
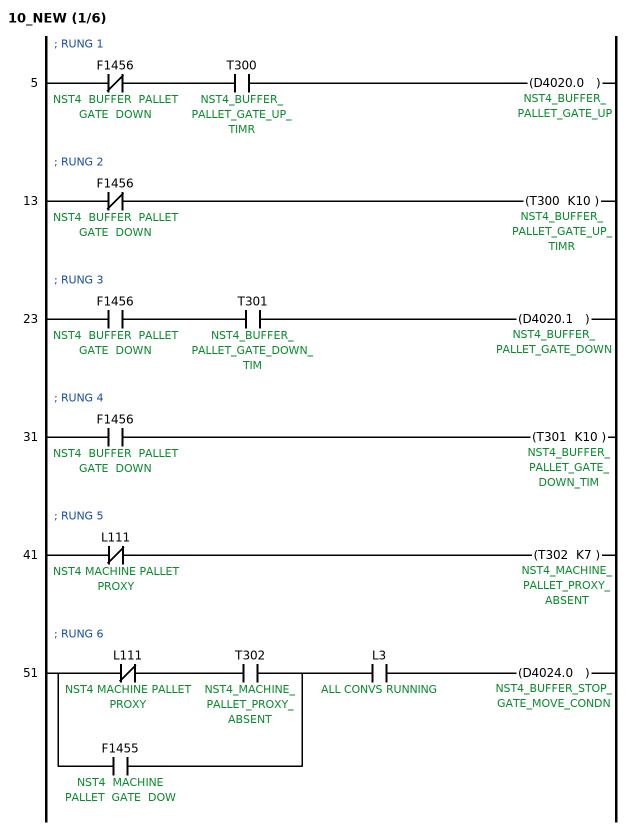
; RUNG 1
5     LDI     F1456  ; NST4  BUFFER  PALLET  GATE  DOWN
      AND     T300  ; NST4_BUFFER_PALLET_GATE_UP_TIMR
      OUT     D4020.0  ; NST4_BUFFER_PALLET_GATE_UP
; RUNG 2
13    LDI     F1456  ; NST4  BUFFER  PALLET  GATE  DOWN
      OUT     T300 K10  ; NST4_BUFFER_PALLET_GATE_UP_TIMR
; RUNG 3
23    LD      F1456  ; NST4  BUFFER  PALLET  GATE  DOWN
      AND     T301  ; NST4_BUFFER_PALLET_GATE_DOWN_TIM
      OUT     D4020.1  ; NST4_BUFFER_PALLET_GATE_DOWN
; RUNG 4
31    LD      F1456  ; NST4  BUFFER  PALLET  GATE  DOWN
      OUT     T301 K10  ; NST4_BUFFER_PALLET_GATE_DOWN_TIM
; RUNG 5
41    LDI     L111  ; NST4 MACHINE PALLET PROXY
      OUT     T302 K7  ; NST4_MACHINE_PALLET_PROXY_ABSENT
; RUNG 6
51    LDI     L111  ; NST4 MACHINE PALLET PROXY
      AND     T302  ; NST4_MACHINE_PALLET_PROXY_ABSENT
      OR      F1455  ; NST4  MACHINE  PALLET  GATE  DOW
      AND     L3  ; ALL CONVS RUNNING
      OUT     D4024.0  ; NST4_BUFFER_STOP_GATE_MOVE_CONDN
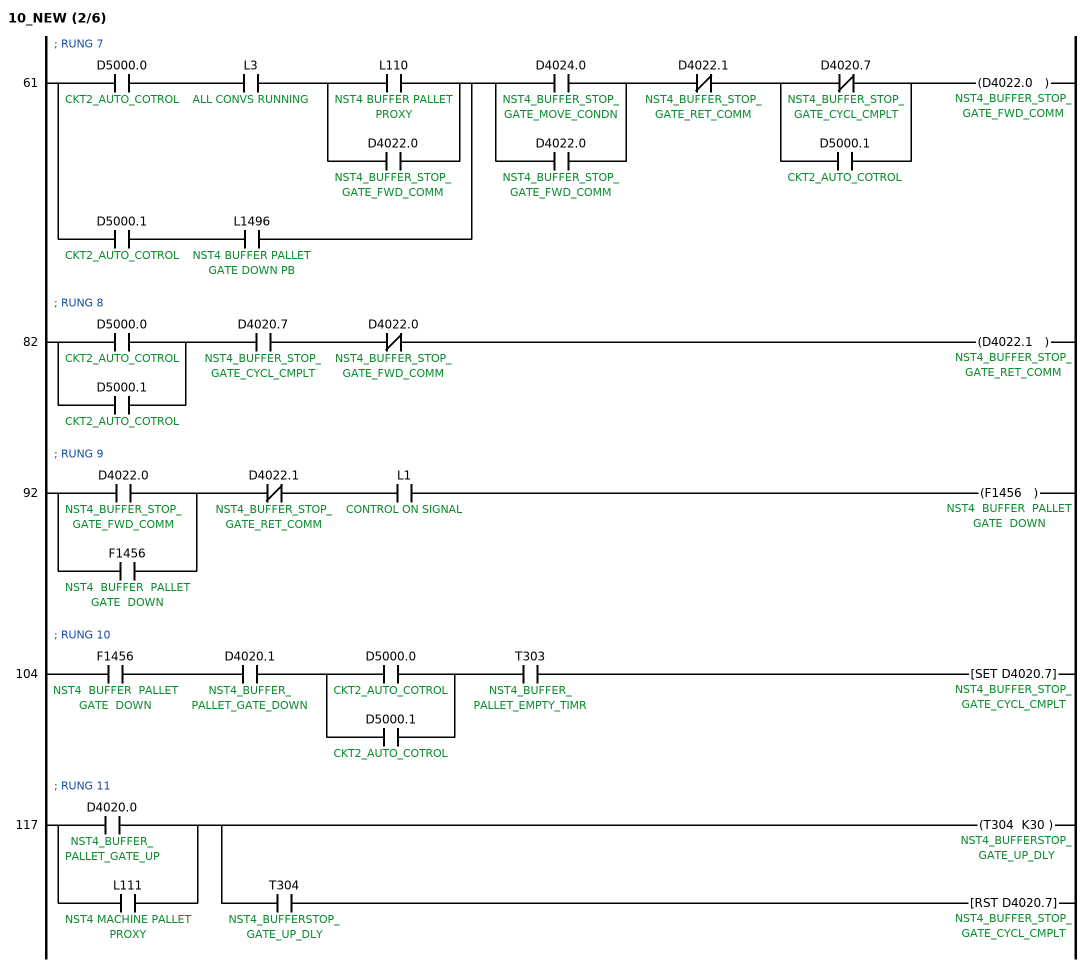
; RUNG 7
61    LD      D5000.0  ; CKT2_AUTO_COTROL
      AND     L3  ; ALL CONVS RUNNING
      LD      L110  ; NST4 BUFFER PALLET PROXY
      OR      D4022.0  ; NST4_BUFFER_STOP_GATE_FWD_COMM
      ANB
      LD      D5000.1  ; CKT2_AUTO_COTROL
      AND     L1496  ; NST4 BUFFER PALLET GATE DOWN PB
      ORB
      LD      D4024.0  ; NST4_BUFFER_STOP_GATE_MOVE_CONDN
      OR      D4022.0  ; NST4_BUFFER_STOP_GATE_FWD_COMM
      ANB
      ANI     D4022.1  ; NST4_BUFFER_STOP_GATE_RET_COMM
      LDI     D4020.7  ; NST4_BUFFER_STOP_GATE_CYCL_CMPLT
      OR      D5000.1  ; CKT2_AUTO_COTROL
      ANB
      OUT     D4022.0  ; NST4_BUFFER_STOP_GATE_FWD_COMM
; RUNG 8
82    LD      D5000.0  ; CKT2_AUTO_COTROL
      OR      D5000.1  ; CKT2_AUTO_COTROL
      AND     D4020.7  ; NST4_BUFFER_STOP_GATE_CYCL_CMPLT
      ANI     D4022.0  ; NST4_BUFFER_STOP_GATE_FWD_COMM
      OUT     D4022.1  ; NST4_BUFFER_STOP_GATE_RET_COMM
; RUNG 9
92    LD      D4022.0  ; NST4_BUFFER_STOP_GATE_FWD_COMM
      OR      F1456  ; NST4  BUFFER  PALLET  GATE  DOWN
      ANI     D4022.1  ; NST4_BUFFER_STOP_GATE_RET_COMM
      AND     L1  ; CONTROL ON SIGNAL
      OUT     F1456  ; NST4  BUFFER  PALLET  GATE  DOWN
; RUNG 10
104   LD      F1456  ; NST4  BUFFER  PALLET  GATE  DOWN
      AND     D4020.1  ; NST4_BUFFER_PALLET_GATE_DOWN
      LD      D5000.0  ; CKT2_AUTO_COTROL
      OR      D5000.1  ; CKT2_AUTO_COTROL
      ANB
      AND     T303  ; NST4_BUFFER_PALLET_EMPTY_TIMR
      SET     D4020.7  ; NST4_BUFFER_STOP_GATE_CYCL_CMPLT
; RUNG 11
117   LD      D4020.0  ; NST4_BUFFER_PALLET_GATE_UP
      OR      L111  ; NST4 MACHINE PALLET PROXY
      OUT     T304 K30  ; NST4_BUFFERSTOP_GATE_UP_DLY
      AND     T304  ; NST4_BUFFERSTOP_GATE_UP_DLY
      RST     D4020.7  ; NST4_BUFFER_STOP_GATE_CYCL_CMPLT
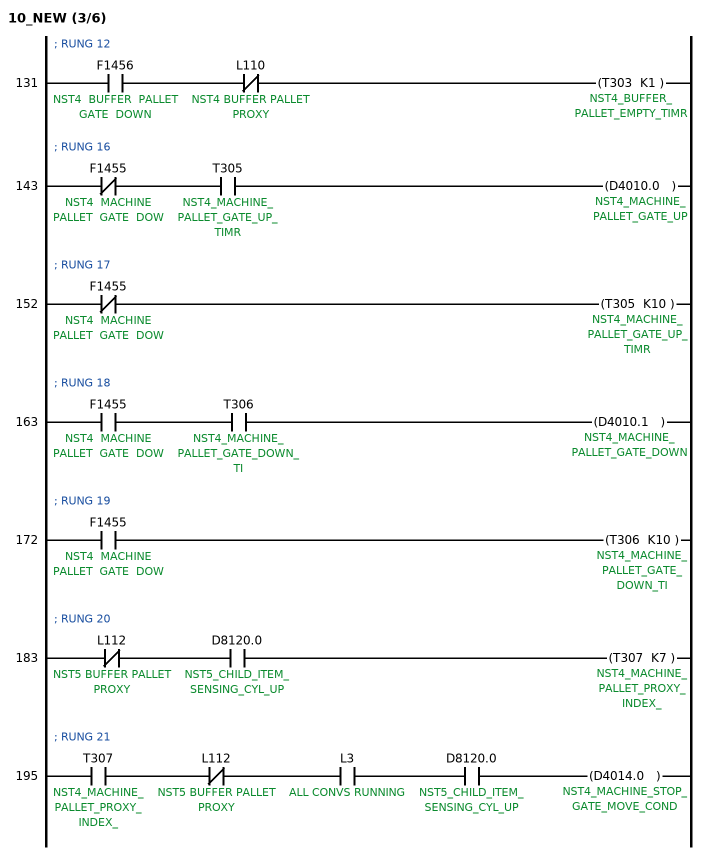
; RUNG 12
131   LD      F1456  ; NST4  BUFFER  PALLET  GATE  DOWN
      ANI     L110  ; NST4 BUFFER PALLET PROXY
      OUT     T303 K1  ; NST4_BUFFER_PALLET_EMPTY_TIMR
; RUNG 16
143   LDI     F1455  ; NST4  MACHINE  PALLET  GATE  DOW
      AND     T305  ; NST4_MACHINE_PALLET_GATE_UP_TIMR
      OUT     D4010.0  ; NST4_MACHINE_PALLET_GATE_UP
; RUNG 17
152   LDI     F1455  ; NST4  MACHINE  PALLET  GATE  DOW
      OUT     T305 K10  ; NST4_MACHINE_PALLET_GATE_UP_TIMR
; RUNG 18
163   LD      F1455  ; NST4  MACHINE  PALLET  GATE  DOW
      AND     T306  ; NST4_MACHINE_PALLET_GATE_DOWN_TI
      OUT     D4010.1  ; NST4_MACHINE_PALLET_GATE_DOWN
; RUNG 19
172   LD      F1455  ; NST4  MACHINE  PALLET  GATE  DOW
      OUT     T306 K10  ; NST4_MACHINE_PALLET_GATE_DOWN_TI
; RUNG 20
183   LDI     L112  ; NST5 BUFFER PALLET PROXY
      AND     D8120.0  ; NST5_CHILD_ITEM_SENSING_CYL_UP
      OUT     T307 K7  ; NST4_MACHINE_PALLET_PROXY_INDEX_
; RUNG 21
195   LD      T307  ; NST4_MACHINE_PALLET_PROXY_INDEX_
      ANI     L112  ; NST5 BUFFER PALLET PROXY
      AND     L3  ; ALL CONVS RUNNING
      AND     D8120.0  ; NST5_CHILD_ITEM_SENSING_CYL_UP
      OUT     D4014.0  ; NST4_MACHINE_STOP_GATE_MOVE_COND
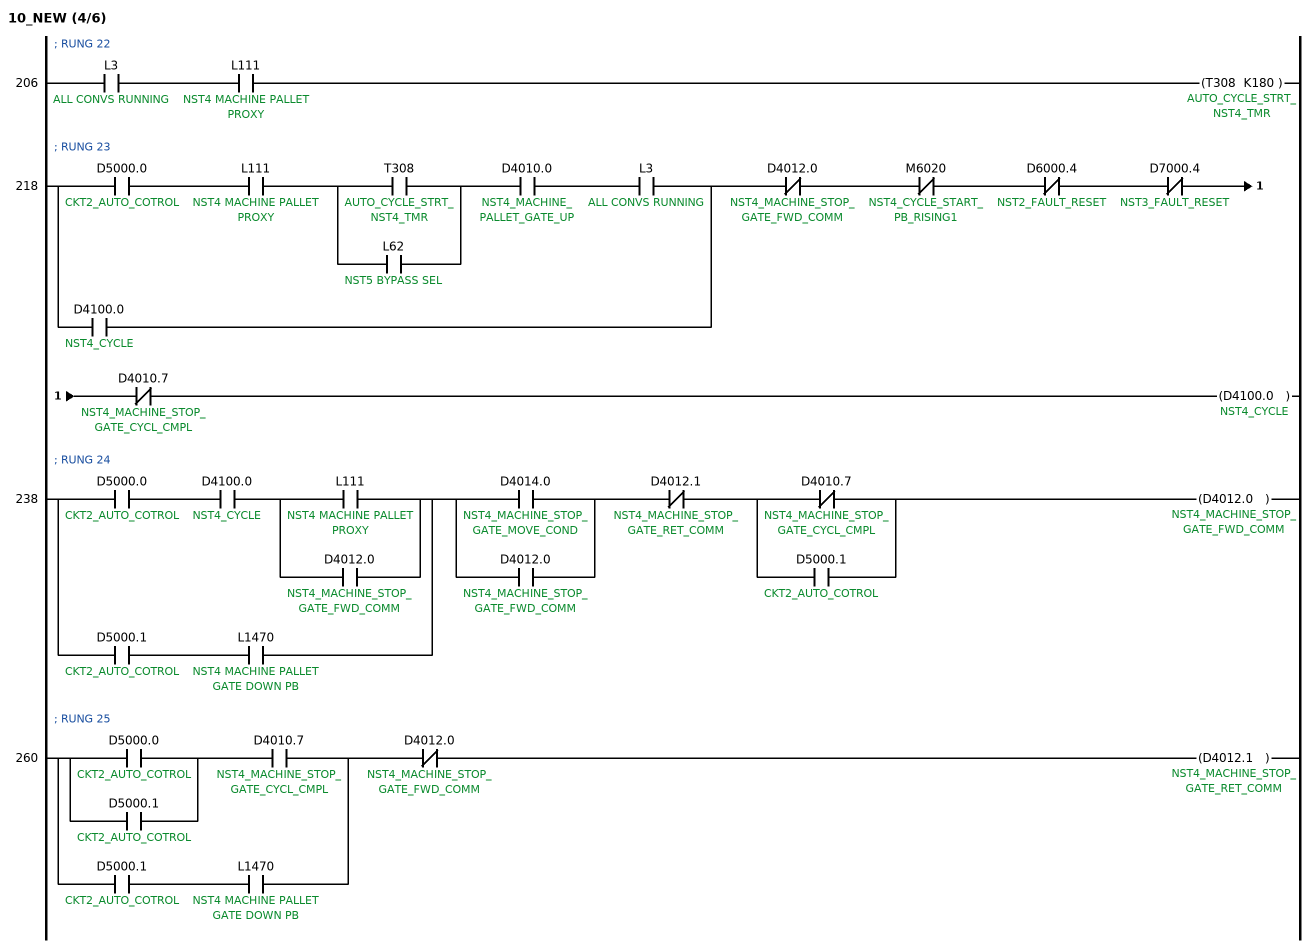
; RUNG 22
206   LD      L3  ; ALL CONVS RUNNING
      AND     L111  ; NST4 MACHINE PALLET PROXY
      OUT     T308 K180  ; AUTO_CYCLE_STRT_NST4_TMR
; RUNG 23
218   LD      D5000.0  ; CKT2_AUTO_COTROL
      AND     L111  ; NST4 MACHINE PALLET PROXY
      LD      T308  ; AUTO_CYCLE_STRT_NST4_TMR
      OR      L62  ; NST5 BYPASS SEL
      ANB
      AND     D4010.0  ; NST4_MACHINE_PALLET_GATE_UP
      AND     L3  ; ALL CONVS RUNNING
      OR      D4100.0  ; NST4_CYCLE
      ANI     D4012.0  ; NST4_MACHINE_STOP_GATE_FWD_COMM
      ANI     M6020  ; NST4_CYCLE_START_PB_RISING1
      ANI     D6000.4  ; NST2_FAULT_RESET
      ANI     D7000.4  ; NST3_FAULT_RESET
      ANI     D4010.7  ; NST4_MACHINE_STOP_GATE_CYCL_CMPL
      OUT     D4100.0  ; NST4_CYCLE
; RUNG 24
238   LD      D5000.0  ; CKT2_AUTO_COTROL
      AND     D4100.0  ; NST4_CYCLE
      LD      L111  ; NST4 MACHINE PALLET PROXY
      OR      D4012.0  ; NST4_MACHINE_STOP_GATE_FWD_COMM
      ANB
      LD      D5000.1  ; CKT2_AUTO_COTROL
      AND     L1470  ; NST4 MACHINE PALLET GATE DOWN PB
      ORB
      LD      D4014.0  ; NST4_MACHINE_STOP_GATE_MOVE_COND
      OR      D4012.0  ; NST4_MACHINE_STOP_GATE_FWD_COMM
      ANB
      ANI     D4012.1  ; NST4_MACHINE_STOP_GATE_RET_COMM
      LDI     D4010.7  ; NST4_MACHINE_STOP_GATE_CYCL_CMPL
      OR      D5000.1  ; CKT2_AUTO_COTROL
      ANB
      OUT     D4012.0  ; NST4_MACHINE_STOP_GATE_FWD_COMM
; RUNG 25
260   LD      D5000.0  ; CKT2_AUTO_COTROL
      OR      D5000.1  ; CKT2_AUTO_COTROL
      AND     D4010.7  ; NST4_MACHINE_STOP_GATE_CYCL_CMPL
      LD      D5000.1  ; CKT2_AUTO_COTROL
      AND     L1470  ; NST4 MACHINE PALLET GATE DOWN PB
      ORB
      ANI     D4012.0  ; NST4_MACHINE_STOP_GATE_FWD_COMM
      OUT     D4012.1  ; NST4_MACHINE_STOP_GATE_RET_COMM
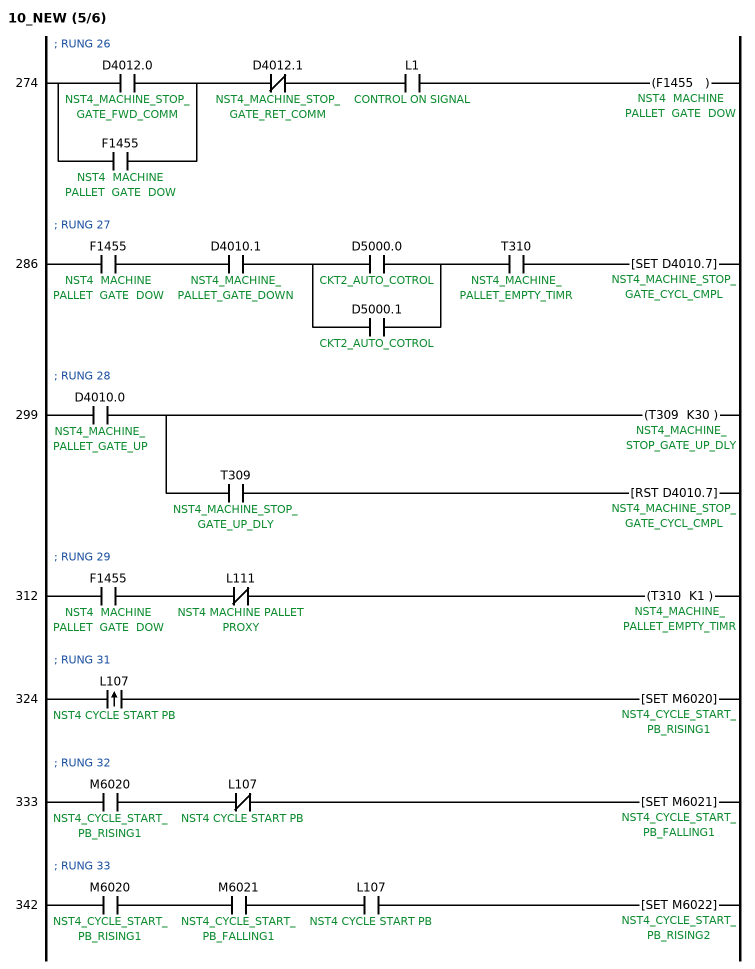
; RUNG 26
274   LD      D4012.0  ; NST4_MACHINE_STOP_GATE_FWD_COMM
      OR      F1455  ; NST4  MACHINE  PALLET  GATE  DOW
      ANI     D4012.1  ; NST4_MACHINE_STOP_GATE_RET_COMM
      AND     L1  ; CONTROL ON SIGNAL
      OUT     F1455  ; NST4  MACHINE  PALLET  GATE  DOW
; RUNG 27
286   LD      F1455  ; NST4  MACHINE  PALLET  GATE  DOW
      AND     D4010.1  ; NST4_MACHINE_PALLET_GATE_DOWN
      LD      D5000.0  ; CKT2_AUTO_COTROL
      OR      D5000.1  ; CKT2_AUTO_COTROL
      ANB
      AND     T310  ; NST4_MACHINE_PALLET_EMPTY_TIMR
      SET     D4010.7  ; NST4_MACHINE_STOP_GATE_CYCL_CMPL
; RUNG 28
299   LD      D4010.0  ; NST4_MACHINE_PALLET_GATE_UP
      OUT     T309 K30  ; NST4_MACHINE_STOP_GATE_UP_DLY
      AND     T309  ; NST4_MACHINE_STOP_GATE_UP_DLY
      RST     D4010.7  ; NST4_MACHINE_STOP_GATE_CYCL_CMPL
; RUNG 29
312   LD      F1455  ; NST4  MACHINE  PALLET  GATE  DOW
      ANI     L111  ; NST4 MACHINE PALLET PROXY
      OUT     T310 K1  ; NST4_MACHINE_PALLET_EMPTY_TIMR
; RUNG 31
324   LDP     L107  ; NST4 CYCLE START PB
      SET     M6020  ; NST4_CYCLE_START_PB_RISING1
; RUNG 32
333   LD      M6020  ; NST4_CYCLE_START_PB_RISING1
      ANI     L107  ; NST4 CYCLE START PB
      SET     M6021  ; NST4_CYCLE_START_PB_FALLING1
; RUNG 33
342   LD      M6020  ; NST4_CYCLE_START_PB_RISING1
      AND     M6021  ; NST4_CYCLE_START_PB_FALLING1
      AND     L107  ; NST4 CYCLE START PB
      SET     M6022  ; NST4_CYCLE_START_PB_RISING2
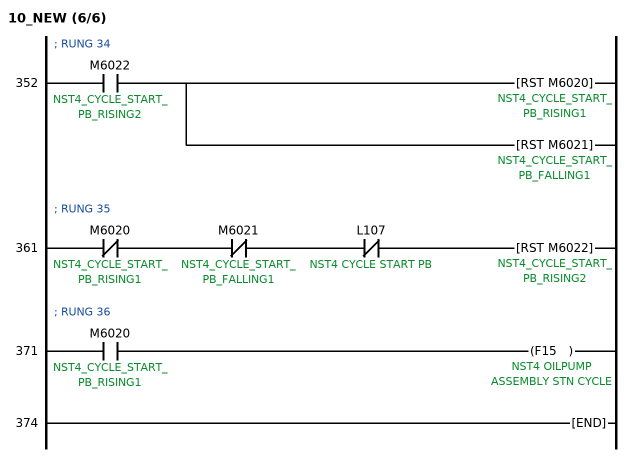
; RUNG 34
352   LD      M6022  ; NST4_CYCLE_START_PB_RISING2
      RST     M6020  ; NST4_CYCLE_START_PB_RISING1
      RST     M6021  ; NST4_CYCLE_START_PB_FALLING1
; RUNG 35
361   LDI     M6020  ; NST4_CYCLE_START_PB_RISING1
      ANI     M6021  ; NST4_CYCLE_START_PB_FALLING1
      ANI     L107  ; NST4 CYCLE START PB
      RST     M6022  ; NST4_CYCLE_START_PB_RISING2
; RUNG 36
371   LD      M6020  ; NST4_CYCLE_START_PB_RISING1
      OUT     F15  ; NST4 OILPUMP ASSEMBLY STN CYCLE
374   END
END_PROGRAM

PROGRAM 11_NEW  // ST5 CK2
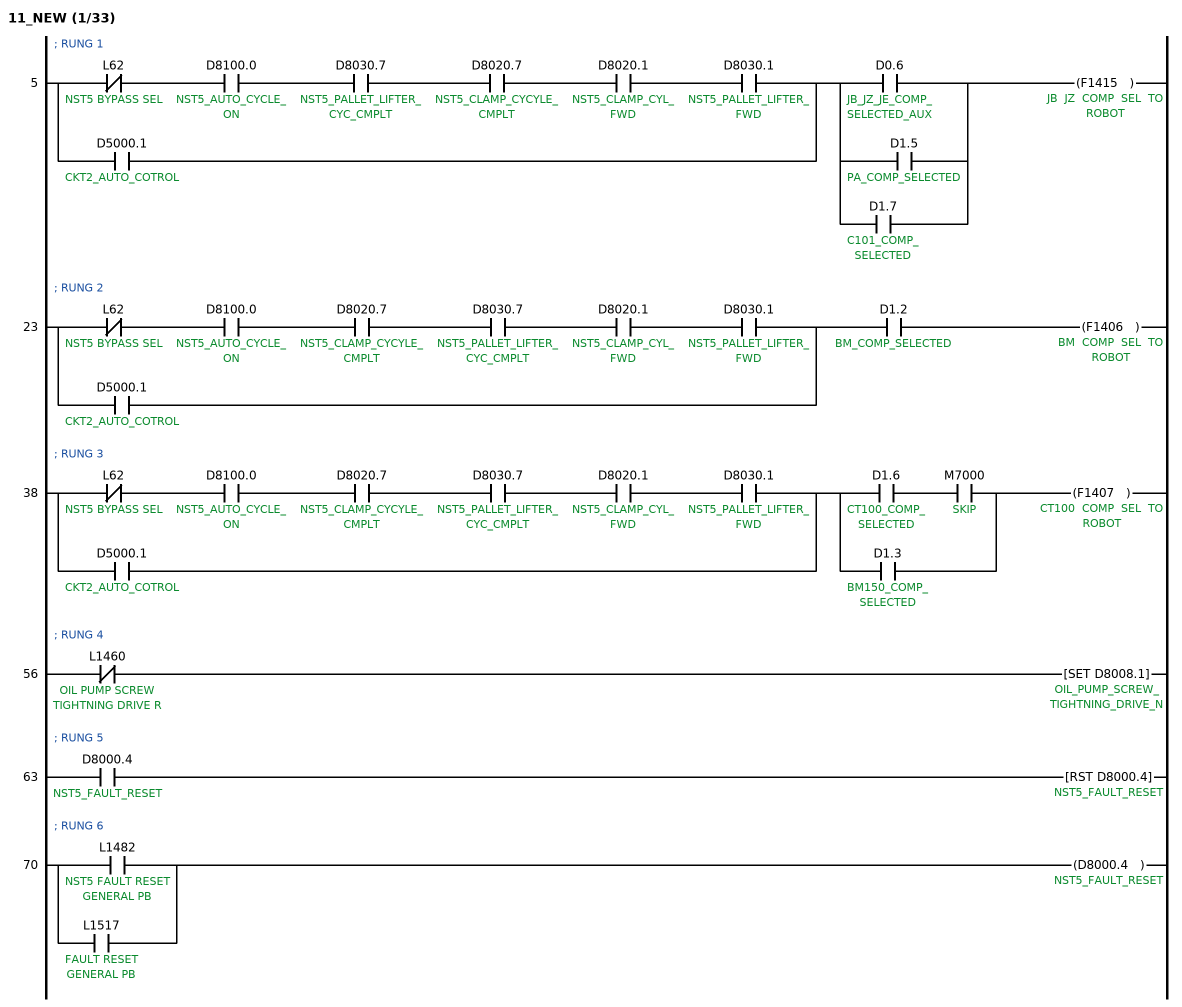
; RUNG 1
5     LDI     L62  ; NST5 BYPASS SEL
      AND     D8100.0  ; NST5_AUTO_CYCLE_ON
      AND     D8030.7  ; NST5_PALLET_LIFTER_CYC_CMPLT
      AND     D8020.7  ; NST5_CLAMP_CYCYLE_CMPLT
      AND     D8020.1  ; NST5_CLAMP_CYL_FWD
      AND     D8030.1  ; NST5_PALLET_LIFTER_FWD
      OR      D5000.1  ; CKT2_AUTO_COTROL
      LD      D0.6  ; JB_JZ_JE_COMP_SELECTED_AUX
      OR      D1.5  ; PA_COMP_SELECTED
      OR      D1.7  ; C101_COMP_SELECTED
      ANB
      OUT     F1415  ; JB  JZ  COMP  SEL  TO  ROBOT
; RUNG 2
23    LDI     L62  ; NST5 BYPASS SEL
      AND     D8100.0  ; NST5_AUTO_CYCLE_ON
      AND     D8020.7  ; NST5_CLAMP_CYCYLE_CMPLT
      AND     D8030.7  ; NST5_PALLET_LIFTER_CYC_CMPLT
      AND     D8020.1  ; NST5_CLAMP_CYL_FWD
      AND     D8030.1  ; NST5_PALLET_LIFTER_FWD
      OR      D5000.1  ; CKT2_AUTO_COTROL
      AND     D1.2  ; BM_COMP_SELECTED
      OUT     F1406  ; BM  COMP  SEL  TO  ROBOT
; RUNG 3
38    LDI     L62  ; NST5 BYPASS SEL
      AND     D8100.0  ; NST5_AUTO_CYCLE_ON
      AND     D8020.7  ; NST5_CLAMP_CYCYLE_CMPLT
      AND     D8030.7  ; NST5_PALLET_LIFTER_CYC_CMPLT
      AND     D8020.1  ; NST5_CLAMP_CYL_FWD
      AND     D8030.1  ; NST5_PALLET_LIFTER_FWD
      OR      D5000.1  ; CKT2_AUTO_COTROL
      LD      D1.6  ; CT100_COMP_SELECTED
      AND     M7000  ; SKIP
      OR      D1.3  ; BM150_COMP_SELECTED
      ANB
      OUT     F1407  ; CT100  COMP  SEL  TO  ROBOT
; RUNG 4
56    LDI     L1460  ; OIL PUMP SCREW TIGHTNING DRIVE R
      SET     D8008.1  ; OIL_PUMP_SCREW_TIGHTNING_DRIVE_N
; RUNG 5
63    LD      D8000.4  ; NST5_FAULT_RESET
      RST     D8000.4  ; NST5_FAULT_RESET
; RUNG 6
70    LD      L1482  ; NST5 FAULT RESET GENERAL PB
      OR      L1517  ; FAULT RESET GENERAL PB
      OUT     D8000.4  ; NST5_FAULT_RESET
